FUNCTION_BLOCK ABSTRACT CollectionEventHandlerBase IMPLEMENTS I_EventHandler
VAR
	_eventReceived : BOOL;
	fromExpected : BOOL;
END_VAR

PROPERTY PUBLIC EventReceived : BOOL
GET // PUBLIC
EventReceived := _eventReceived;
END_GET
END_PROPERTY

PROPERTY PUBLIC FromExpectedOriginator : BOOL
GET // PUBLIC
FromExpectedOriginator := fromExpected;
END_GET
END_PROPERTY

METHOD PUBLIC ABSTRACT HandleEvent
VAR_INPUT
	Event : I_Event;
END_VAR
END_METHOD

METHOD PUBLIC Reset
_eventReceived := FALSE;
fromExpected := FALSE;
END_METHOD

END_FUNCTION_BLOCK

(* stored: Version 1.1.0.1, ProductVersion 3.1.4024.12
   POU CollectionEventHandlerBase: Id {a239ba6b-4188-09cd-395e-cbbd0ad7e8a5}, SpecialFunc None
   Property EventReceived: Id {de345d68-3ace-0ebc-2649-ceb58b6cda03}
   Get Get: Id {9f1a9e6a-e9e4-025a-169b-0c5a68074274}
   Property FromExpectedOriginator: Id {93038ab0-2de4-07ac-146b-365f02981392}
   Get Get: Id {43da309a-5f87-0cce-3b82-1e3e844574f8}
   Method HandleEvent: Id {12fdce4e-65e8-06a3-3a33-d475f14d5e54}
   Method Reset: Id {c2830d50-934a-0ce2-325a-095eb6036186} *)
